(* CoDeSys 2.3 export: FLE.EXP *)

(* Data type in BathFB *)
TYPE FlE :
(
    NoFl,    (*нет жидкости*)
    TMS,
    water
);
END_TYPE
